TYPE UR_9_O2T_Ints :
STRUCT
      Ints : ARRAY[0..11] OF DINT;
END_STRUCT
END_TYPE

(* stored: Version 1.1.0.1
   DUT UR_9_O2T_Ints: Id {3f9fd3a2-c8a1-4ba8-8832-fc66f7b37eb6} *)
